SUBAPPLICATION GreenWhiteBackground3C (* Hintergrundfarbe (TRUE -> Grün, FALSE -> Weiß) für 3 Objekte (Kompakt) *)
  (* Standard: 61499-2 *)
  (* Version 1.0, 2023-02-06, franz, Meisterschulen am Ostbahnhof *)
  PACKAGE MyLib::sys;
  IMPORT isobus::UT::Q::const::IDs::ID_NULL;
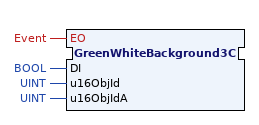
  EVENT_INPUT
    EO;
  END_EVENT
  VAR_INPUT
    DI : BOOL;
    u16ObjId : UINT := ID_NULL;
    u16ObjIdA : UINT;
  END_VAR
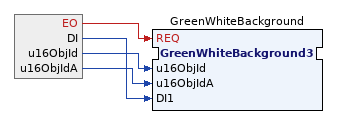
  SUBAPPS
    GreenWhiteBackground : MyLib::sys::GreenWhiteBackground3;
  END_SUBAPPS
  EVENT_CONNECTIONS
    EO TO GreenWhiteBackground.REQ;
  END_CONNECTIONS
  DATA_CONNECTIONS
    u16ObjId TO GreenWhiteBackground.u16ObjId;
    u16ObjIdA TO GreenWhiteBackground.u16ObjIdA;
    DI TO GreenWhiteBackground.DI1;
  END_CONNECTIONS
END_SUBAPPLICATION
